PROGRAM INTERNAL MAIN_TESTS
VAR
	_taskTests : fbTaskTests;
END_VAR

_taskTests();

END_PROGRAM

(* stored: Version 1.1.0.1, ProductVersion 3.1.4024.5
   POU MAIN_TESTS: Id {eacdc333-c1f6-40c7-b492-980a45633e39}, SpecialFunc None *)
